FUNCTION_BLOCK DoorController
  (* Standard: 61499-2 *)
  (* Version 0.1, 2016-00-28, hpea485, UOA *)
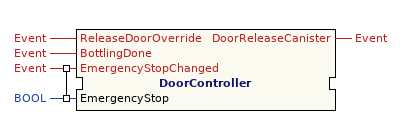
  EVENT_INPUT
    ReleaseDoorOverride;
    BottlingDone;
    EmergencyStopChanged WITH EmergencyStop;
  END_EVENT
  EVENT_OUTPUT
    DoorReleaseCanister;
  END_EVENT
  VAR_INPUT
    EmergencyStop : BOOL;
  END_VAR
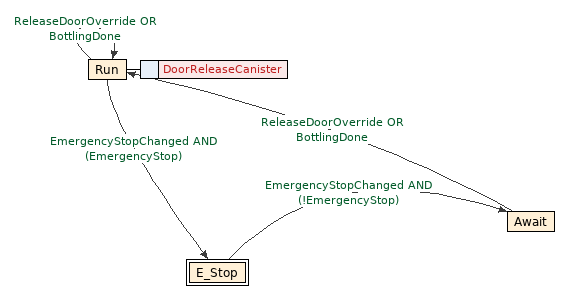
  EC_STATES
    E_Stop;
    Run : -> DoorReleaseCanister;
    Await;
  END_STATES
  EC_TRANSITIONS
    Run TO E_Stop := EmergencyStopChanged AND (EmergencyStop);
    Run TO Run := ReleaseDoorOverride OR BottlingDone;
    E_Stop TO Await := EmergencyStopChanged AND (!EmergencyStop);
    Await TO Run := ReleaseDoorOverride OR BottlingDone;
  END_TRANSITIONS
END_FUNCTION_BLOCK
